// TwinCAT 3 PLC project CommInterfaces
// ProgramVersion: 3.1.4026.12
// libraries:
//   Tc2_ModbusSrv, * (Beckhoff Automation GmbH)
//   Tc2_Standard, * (Beckhoff Automation GmbH)
//   Tc2_System, * (Beckhoff Automation GmbH)
//   Tc2_Utilities, * (Beckhoff Automation GmbH)
//   Tc3_IotBase, * (Beckhoff Automation GmbH)
//   Tc3_Module, * (Beckhoff Automation GmbH)
//   Tc3_JsonXml,3.3.12.0,Beckhoff Automation GmbH
// project tree:
//   DataTypes/ ControlBESScmds.TcDUT, ControlBESSparams.TcDUT, feederMeteringStruct.TcDUT, feederJSONStruct.TcDUT
//   GVLs/ metering.TcGVL
//   / MQTTPub.TcTTO, MQTTSub.TcTTO, ReadFD083.TcTTO
//   Program/ MQTTPublish.TcPOU, ModbusRead.TcPOU, MQTTSubscribe.TcPOU
//   Utils/ FB_MakeTimestamp.TcPOU, FUN_LeftZeroPadding.TcPOU
// real-time tasks:
//   TASK ReadFD083: cycle T#10ms, priority 1, ADS port 351
//   TASK MQTTPub: cycle T#1ms, priority 3, ADS port 352
//   TASK MQTTSub: cycle T#10ms, priority 2, ADS port 353

CONFIGURATION CommInterfaces
    RESOURCE PLC ON TwinCAT3
        TASK MQTTPub(INTERVAL := T#1ms, PRIORITY := 3);
        TASK MQTTSub(INTERVAL := T#10ms, PRIORITY := 2);
        TASK ReadFD083(INTERVAL := T#10ms, PRIORITY := 1);
        PROGRAM MQTTSubscribe WITH MQTTSub : MQTTSubscribe;
        PROGRAM ModbusRead WITH ReadFD083 : ModbusRead;
    END_RESOURCE
END_CONFIGURATION

// ---- DataTypes/ControlBESScmds.TcDUT
TYPE ControlBESScmds :
STRUCT
	start: BOOL;
END_STRUCT
END_TYPE

// ---- DataTypes/ControlBESSparams.TcDUT
TYPE ControlBESSparams :
STRUCT
END_STRUCT
END_TYPE

// ---- DataTypes/feederMeteringStruct.TcDUT
{attribute 'pack_mode' := '1'} 
TYPE feederMeteringStruct :
STRUCT
	YEAR                   			: INT; //0
	MONTH 							: INT; //2
	DAY 							: INT; //4
	HOUR 							: INT; //6
	MINUTE 							: INT; //8
	SECOND 							: INT; //10
	
	PV_GENERATION_kW 				: INT; // SCALED by 1000
	TOTAL_APPARENT_LOAD_POWER_kVA	: INT; // SCALED by 1000
	LOAD_P_kW						: INT;
	VOLTAGE_MIN_pu					: INT;
	VOLTAGE_MAX_pu					: INT;
	LOADING_MAX						: INT;
	LOADING_MIN						: INT;
	VOLTAGE_DROP_MAX				: INT;
	VOLTAGE_DROP_MIN				: INT;
	GENERATION_ACTIVE_POWER_kW		: INT;
	INFEED_ACTIVE_POWER_kW			: INT;
	TOTAL_LOAD_P_kW					: INT;
	LOSSES_kW						: INT;
END_STRUCT
END_TYPE

// ---- DataTypes/feederJSONStruct.TcDUT
TYPE feederJSONStruct :
STRUCT
	TIMESTAMP : STRING;
	PV_GENERATION_kW 				: REAL;
	TOTAL_APPARENT_LOAD_POWER_kVA	: REAL; 
	VOLTAGE_MIN_pu					: REAL;
	VOLTAGE_MAX_pu					: REAL;
	LOADING_MAX						: REAL;
	LOADING_MIN						: REAL;
	VOLTAGE_DROP_MAX				: REAL;
	VOLTAGE_DROP_MIN				: REAL;
	GENERATION_ACTIVE_POWER_kW		: REAL;
	INFEED_ACTIVE_POWER_kW			: REAL;
	TOTAL_LOAD_P_kW					: REAL;
	LOSSES_kW						: REAL;
END_STRUCT
END_TYPE

// ---- GVLs/metering.TcGVL
{attribute 'qualified_only'}
VAR_GLOBAL
	//metering signals
		MeteringSignals : feederMeteringStruct;
END_VAR

// ---- Program/MQTTSubscribe.TcPOU
PROGRAM MQTTSubscribe
VAR
    (* received payload for each subscribed topic *)
	{attribute 'TcEncoding':='UTF-8'}
    sPayloadRcv1 : STRING(255);
	//{attribute 'TcEncoding':='UTF-8'}
    sPayloadRcv2 : STRING(255);
	
    fbMessageQueue 	: FB_IotMqttMessageQueue;
    fbMessage     	: FB_IotMqttMessage;
	fbMqttClient    : FB_IotMqttClient;
	
    bSetParameter   : BOOL := TRUE;
    bConnect        : BOOL := TRUE;
	bSubscribed     : ARRAY[1..2] OF BOOL;
	
	i: INT;
	noOfTopics: INT:= 2;
	
END_VAR
VAR CONSTANT
    (* subscriptions *)
    sTopicSub1 : STRING(255) := 'Feeder/BESS/control/commands';
    sTopicSub2 : STRING(255) := 'Feeder/BESS/control/params'; 
	
	sTopicSub : ARRAY [1..2] OF STRING:=[sTopicSub1, sTopicSub1];
END_VAR

IF bSetParameter THEN
	bSetParameter				:= FALSE;
    fbMqttClient.sHostName 		:= 'a3rq4sh4gv4om5-ats.iot.eu-west-3.amazonaws.com'; 
    fbMqttClient.nHostPort 		:= 8883;
    fbMqttClient.sTopicPrefix 	:= '';
    fbMqttClient.sClientId 		:= 'PLC1';
  	fbMqttClient.stTLS.sCA 		:= 'C:\Users\tecnicoloyolatech\Desktop\certs\AmazonRootCA1.pem';
  	fbMqttClient.stTLS.sCert 	:= 'C:\Users\tecnicoloyolatech\Desktop\certs\b729f5b134b28288523e0bb227f630967d68e270326ba912b4ddb8638ad6c3c6-certificate.pem.crt';
  	fbMqttClient.stTLS.sKeyFile := 'C:\Users\tecnicoloyolatech\Desktop\certs\b729f5b134b28288523e0bb227f630967d68e270326ba912b4ddb8638ad6c3c6-private.pem.key';
  	fbMqttClient.ActivateExponentialBackoff(T#1S, T#30S);
	fbMqttClient.ipMessageQueue := fbMessageQueue;
	//FOR i:= 1 TO noOfTopics DO
	//	bSubscribed[i] := fbMqttClient.Subscribe(sTopic:=sTopicSub[i], eQoS:=TcIotMqttQos.AtMostOnceDelivery);
	//END_FOR
END_IF


fbMqttClient.Execute(bConnect);
fbMqttClient.bConnected;
fbMqttClient.hrErrorCode;
fbMqttClient.eConnectionState;
IF fbMessageQueue.nQueuedMessages > 0 THEN

    IF fbMessageQueue.Dequeue(fbMessage:=fbMessage) THEN
        IF fbMessage.CompareTopic(sTopic:=sTopicSub1) THEN
            fbMessage.GetPayload(pPayload:=ADR(sPayloadRcv1), nPayloadSize:=SIZEOF(sPayloadRcv1), bSetNullTermination:=FALSE);
        ELSIF fbMessage.CompareTopic(sTopic:=sTopicSub2) THEN
            fbMessage.GetPayload(pPayload:=ADR(sPayloadRcv2), nPayloadSize:=SIZEOF(sPayloadRcv2), bSetNullTermination:=FALSE);
        END_IF
    END_IF
END_IF

END_PROGRAM

// ---- Program/ModbusRead.TcPOU
PROGRAM ModbusRead
VAR
	
	datetimeVector : ARRAY [1 .. 6] OF INT;
	signalsVector: ARRAY [1 .. 13] OF REAL;
	scale : REAL := 1000.0;
	
	ipAddr    		: STRING(15) := '10.30.244.10'; // ModbusServer
	ipAddrPort		: UINT := 12345;
	
	//Feeder FD_083
	fbReadRegs	:	FB_MBReadRegs;
	mbreadcounter	:	INT;


END_VAR

IF (NOT fbReadRegs.bBusy) THEN
	fbReadRegs(bExecute:=TRUE,
			   sIPAddr := ipAddr,
			   nTCPPort := ipAddrPort,
			   nQuantity := SIZEOF(metering.MeteringSignals)/2,
		       nMBAddr := 0,
			   cbLength := SIZEOF(metering.MeteringSignals),
			   pDestAddr := ADR(metering.MeteringSignals),
			   tTimeout := T#10S,
			   nUnitID := 16#FF); 
ELSE 
	fbReadRegs(bExecute:=FALSE);
END_IF
	
// Assign the vectorized timestamp in the datatimeVector ARRAY
datetimeVector[1] := metering.MeteringSignals.YEAR;
datetimeVector[2] := metering.MeteringSignals.MONTH;
datetimeVector[3] := metering.MeteringSignals.DAY;
datetimeVector[4] := metering.MeteringSignals.HOUR;
datetimeVector[5] := metering.MeteringSignals.MINUTE;
datetimeVector[6] := metering.MeteringSignals.SECOND;

// Assign the incoming metering signas to meteringSignals ARRAY
signalsVector[1] := metering.MeteringSignals.PV_GENERATION_kW/scale;
signalsVector[2] := metering.MeteringSignals.TOTAL_APPARENT_LOAD_POWER_kVA/scale;
signalsVector[3] := metering.MeteringSignals.LOAD_P_kW/scale;
signalsVector[4] := metering.MeteringSignals.VOLTAGE_MIN_pu/scale;
signalsVector[5] := metering.MeteringSignals.VOLTAGE_MAX_pu/scale;
signalsVector[6] := metering.MeteringSignals.LOADING_MAX/scale;
signalsVector[7] := metering.MeteringSignals.LOADING_MIN/scale;
signalsVector[8] := metering.MeteringSignals.VOLTAGE_DROP_MAX/scale;
signalsVector[9] := metering.MeteringSignals.VOLTAGE_DROP_MIN/scale;
signalsVector[10] := metering.MeteringSignals.GENERATION_ACTIVE_POWER_kW/scale;
signalsVector[11] := metering.MeteringSignals.INFEED_ACTIVE_POWER_kW/scale;
signalsVector[12] := metering.MeteringSignals.TOTAL_LOAD_P_kW/scale;
signalsVector[13] := metering.MeteringSignals.LOSSES_kW/scale;

END_PROGRAM

// ---- Program/MQTTPublish.TcPOU
PROGRAM MQTTPublish
VAR
	fbMqttClient: FB_IotMqttClient; // MQTT client.
	fbJsonDataType : FB_JsonReadWriteDataType;
	fbJson : FB_JsonSaxWriter;
	
	TopicToPublish : STRING(255) := 'Feeder/083';
	sJsonDoc : STRING(255); //String to send in JSON format
	
	fbSendMessageIntervalTimer : TON := (PT:=T#5S);
	fbMakeTimestamp : FB_MakeTimestamp;
	
	scale : REAL := 1000.0;
	bSetParameter   : BOOL := TRUE;
	bConnect        : BOOL := TRUE;	
END_VAR

IF bSetParameter THEN
	bSetParameter				:= FALSE;
    fbMqttClient.sHostName 		:= 'a3rq4sh4gv4om5-ats.iot.eu-west-3.amazonaws.com'; 
    fbMqttClient.nHostPort 		:= 8883;
    fbMqttClient.sTopicPrefix 	:= '';
    fbMqttClient.sClientId 		:= 'PLC1';
  	fbMqttClient.stTLS.sCA 		:= 'C:\Users\tecnicoloyolatech\Desktop\certs\AmazonRootCA1.pem';
  	fbMqttClient.stTLS.sCert 	:= 'C:\Users\tecnicoloyolatech\Desktop\certs\4bcd27ad01e301288efa95a347e67a3ace65b850d1b0ed954ddefa5992b51b8b-certificate.pem.crt';
  	fbMqttClient.stTLS.sKeyFile := 'C:\Users\tecnicoloyolatech\Desktop\certs\4bcd27ad01e301288efa95a347e67a3ace65b850d1b0ed954ddefa5992b51b8b-private.pem.key';
  	fbMqttClient.ActivateExponentialBackoff(T#1S, T#30S);
END_IF

// Keep the connection alive by invoking the Execute on every execution cycle.
fbMqttClient.Execute(bConnect);

// -------------------- Publish ---------------------------------

// If the connection with the MQTT broker is establish
IF fbMqttClient.bConnected THEN
    fbSendMessageIntervalTimer(IN:=TRUE);
    IF fbSendMessageIntervalTimer.Q THEN
        fbSendMessageIntervalTimer(IN:=FALSE);
		
		// Convert signals into a timestamp
		fbMakeTimestamp.year := metering.MeteringSignals.YEAR;
		fbMakeTimestamp.month := metering.MeteringSignals.MONTH;
		fbMakeTimestamp.day:= metering.MeteringSignals.DAY;
		fbMakeTimestamp.hour:= metering.MeteringSignals.HOUR;
		fbMakeTimestamp.minute:= metering.MeteringSignals.MINUTE;
		fbMakeTimestamp.second:= metering.MeteringSignals.SECOND;
		
		fbMakeTimestamp();
		
		// Make the JSON message
		fbJson.StartObject();
		fbJson.AddKey('Timestamp');
		fbJson.AddDateTime(fbMakeTimestamp.timestamp);
		//fbJson.AddKey('Values');
		//fbJson.StartObject();
		fbJson.AddKey('PV Generation (kW)');
		fbJson.AddReal(metering.MeteringSignals.PV_GENERATION_kW/scale);
		fbJson.AddKey('Total Load Power (kVA)');
		fbJson.AddReal(metering.MeteringSignals.TOTAL_APPARENT_LOAD_POWER_kVA/scale);
		fbJson.AddKey('Minimum Terminal Voltage (pu)');
		fbJson.AddReal(metering.MeteringSignals.VOLTAGE_MIN_pu/scale);
		fbJson.AddKey('Maximum Terminal Voltage (pu)');
		fbJson.AddReal(metering.MeteringSignals.VOLTAGE_MAX_pu/scale);
		//fbJson.EndObject();
		fbJson.EndObject();
		sJsonDoc := fbJson.GetDocument();
		fbJson.ResetDocument();
		
     	// Publish message 
        fbMqttClient.Publish(sTopic:= TopicToPublish,
            pPayload:= ADR(sJsonDoc),
            nPayloadSize:= LEN2(ADR(sJsonDoc)),
            eQoS:= TcIotMqttQos.AtMostOnceDelivery,
            bRetain:= FALSE,
            bQueue:= FALSE);
    END_IF
END_IF

END_PROGRAM

// ---- Utils/FB_MakeTimestamp.TcPOU
FUNCTION_BLOCK FB_MakeTimestamp
VAR_INPUT
	year:INT;
	month:INT;
	day:INT;
	hour:INT;
	minute:INT;
	second:INT;
END_VAR
VAR_OUTPUT
	timestamp: DT;
END_VAR
VAR
	temp: STRING(255);
END_VAR

// Start with year i.e. XXXX-
temp:= CONCAT(INT_TO_STRING(year), '-');

// Append the month (in case of a single digit pad with zero) i.e. XXXX-XX-	
temp:= CONCAT(CONCAT(temp, FUN_LeftZeroPadding(month)), '-');

// Append the day (in case of a single digit pad with zero) i.e. XXXX-XX-XX 	
temp:= CONCAT(CONCAT(temp, FUN_LeftZeroPadding(day)), '-');

// Append the hour (in case of a single digit pad with zero) i.e. XXXX-XX-XX XX:
temp:= CONCAT(CONCAT(temp, FUN_LeftZeroPadding(hour)), ':');

// Append the minutes (in case of a single digit pad with zero) i.e. XXXX-XX-XX XX:XX:
temp:= CONCAT(CONCAT(temp, FUN_LeftZeroPadding(minute)), ':');

// Append the seconds  (in case of a single digit pad with zero) i.e. XXXX-XX-XX XX:XX:XX
temp:= CONCAT(temp, FUN_LeftZeroPadding(second));

timestamp:= STRING_TO_DT(CONCAT('DT#', temp));

END_FUNCTION_BLOCK

// ---- Utils/FUN_LeftZeroPadding.TcPOU
FUNCTION FUN_LeftZeroPadding : STRING
VAR_INPUT
	input_string : INT;
END_VAR
VAR
	temp : STRING(255);
END_VAR

temp := INT_TO_STRING(input_string);

IF LEN(temp) = 1 THEN
	FUN_LeftZeroPadding:= CONCAT('0', temp);
ELSIF LEN(temp) = 2 THEN
	FUN_LeftZeroPadding:= temp;
END_IF

END_FUNCTION
